PROGRAM MAIN
VAR
	x : INT;
END_VAR

x := x + 1;
x := undeclared_name;

END_PROGRAM

(* stored: Version 1.1.0.1, ProductVersion 3.1.4026.18
   POU MAIN: Id {00000000-0000-0000-0000-0000000000b1}, SpecialFunc None *)
